{attribute addProperty BoxType "EK1122-0000-0018"}
{attribute addProperty Id "Beckhoff_EL6xxxsub_EK1100EK1100_179A0949162"}
{attribute addProperty CRC "3333885208"}
{attribute addProperty SizeInBites "16"}
{attribute addProperty SizeInBytes "2"}
TYPE Beckhoff_EL6xxxEK1122_C6B70D18 EXTENDS EK1122_179A0949 :
STRUCT
	{attribute addProperty Name "Beckhoff_EL6xxxsub_EK1100"}
	Beckhoff_EL6xxxsub_EK1100 : EK1100_179A0949;
END_STRUCT
END_TYPE

(* stored: Version 1.2.0.0, ProductVersion 3.1.4024.9
   DUT Beckhoff_EL6xxxEK1122_C6B70D18: Id {16aa1a86-d6c2-4f9c-98ac-6673bb1acd95} *)
